PROGRAM MAIN
VAR
END_VAR

END_PROGRAM

(* stored: Version 1.1.0.1
   POU MAIN: Id {802a3237-5067-47bd-aac0-8ed5af624e75} *)
